(*

.. <legal notes>

legal notes
=================
| SPDX-FileCopyrightText: © 2025 Oleksandr Tiutyk <trofimich@gmail.com>
| SPDX-License-Identifier: LGPL-3.0-only
| For details check: LGPL-3.0-only_

.. _LGPL-3.0-only: https://www.gnu.org/licenses/lgpl-3.0.en.html

.. </legal notes>

*)

{attribute 'no_explicit_call' := 'do not call this function block directly'} 
FUNCTION_BLOCK DeleteDirectory EXTENDS TOF_Tasks.Task IMPLEMENTS IFileSystemTask
VAR
	_ClassName : STRING := __POUNAME();

    _DeleteDirectory : Tc2_System.FB_RemoveDir;	
END_VAR

{attribute 'monitoring' := 'call'}
PROPERTY AmsNetId : Tc2_System.T_AmsNetID
GET
AmsNetId := _DeleteDirectory.sNetId;
END_GET
SET
_DeleteDirectory.sNetId := AmsNetId;
END_SET
END_PROPERTY

{attribute 'monitoring' := 'call'}
PROPERTY ClassName : STRING
GET
ClassName := _ClassName;
END_GET
END_PROPERTY

{attribute 'monitoring' := 'call'}
PROPERTY DirectoryPath : Tc2_System.T_MaxString
GET
DirectoryPath := _DeleteDirectory.sPathName;
END_GET
SET
_DeleteDirectory.sPathName := DirectoryPath;
END_SET
END_PROPERTY

{attribute 'monitoring' := 'call'}
PROPERTY NamespaceName : STRING
GET
NamespaceName := CurrentNamespace.Name;
END_GET
END_PROPERTY

METHOD PROTECTED OnCancel
_DeleteDirectory(bExecute := FALSE);
END_METHOD

METHOD PROTECTED OnRunning 
VAR_INPUT
	startRequest : BOOL;
END_VAR
VAR_OUTPUT
	state : TASK_RUNNING_STATE;
END_VAR
VAR
	propertyNotSpecifiedException :	TOF_Core.DataMemberNotSpecifiedException;
	invalidPathException : InvalidPathException;	
	deleteDirectoryException : TOF_Core.StandardException;
	
	pathErrorMessage : WSTRING(255);
	errorMessageBuilder : TOF_Core.WideStringBuilder;
END_VAR
IF startRequest THEN 
	IF TOF_Core.StringHelper.IsNullOrWhiteSpace(_DeleteDirectory.sPathName) THEN
		propertyNotSpecifiedException.Throw(NamespaceName, ClassName, __POUNAME(), __POSITION(), 'DirectoryPath');		
	END_IF
	
	IF NOT PathHelper.IsValidDirectoryPath(_DeleteDirectory.sPathName, errorMessage => pathErrorMessage) THEN
		invalidPathException.Throw(NamespaceName, ClassName, __POUNAME(), __POSITION(), _DeleteDirectory.sPathName, pathErrorMessage);
	END_IF
	
	_DeleteDirectory(bExecute := FALSE);
END_IF

_DeleteDirectory(bExecute := TRUE);

IF _DeleteDirectory.bError THEN
	errorMessageBuilder
		.AppendString("An error occurred while deleting the directory '")
		.Append(_DeleteDirectory.sPathName)
		.AppendString("'");

	deleteDirectoryException.Throw(NamespaceName, ClassName, __POUNAME(), __POSITION(), errorMessageBuilder.ToString255(), errorCode := _DeleteDirectory.nErrId);
END_IF

IF NOT _DeleteDirectory.bBusy THEN
	state := TOF_Tasks.TASK_RUNNING_STATE.DONE;
END_IF
END_METHOD

{attribute 'monitoring' := 'call'}
PROPERTY PathType : Tc2_System.E_OpenPath
GET
PathType := _DeleteDirectory.ePath;
END_GET
SET
_DeleteDirectory.ePath := PathType;
END_SET
END_PROPERTY

{attribute 'monitoring' := 'call'}
PROPERTY Size : ULINT
GET
Size := XSIZEOF(THIS^);
END_GET
END_PROPERTY

{attribute 'monitoring' := 'call'}
PROPERTY Timeout : TIME
GET
Timeout := _DeleteDirectory.tTimeout;
END_GET
SET
_DeleteDirectory.tTimeout := Timeout;
END_SET
END_PROPERTY

END_FUNCTION_BLOCK

(* stored: Version 1.1.0.1
   POU DeleteDirectory: Id {f7699339-eb16-4c49-8ff9-e8b510a181bf}, SpecialFunc None
   Folder Inputs: Id {3c1b2bb2-508a-43ab-aba6-d51610d36987}
   Folder Members to override: Id {80e81cc0-48cb-4c8d-a6d2-f5019c2649ac}
   Property AmsNetId: Id {e619447a-91f5-4cfd-87c1-c6f4d65469a7}
   Get Get: Id {af838fb5-84a9-40c2-96ed-bb37e1ba8ee8}
   Set Set: Id {955f8a77-cfbb-437a-a3ea-c4c2072c8db2}
   Property ClassName: Id {9bdfd013-5a24-4a24-9847-b8d276cbdfd1}
   Get Get: Id {07f43309-f5f9-4714-8a79-b20e37081f91}
   Property DirectoryPath: Id {d94128c9-a1f4-40bf-a870-d7916c828353}
   Get Get: Id {1f72f3d7-a990-4668-a6c3-c54f2f298ded}
   Set Set: Id {39cb2b34-0284-49a9-954b-190ef76241ef}
   Property NamespaceName: Id {c30ceec4-6b12-4987-9c9a-253d7cedcfe2}
   Get Get: Id {5de19f01-2439-4806-bb38-5c646f83ed28}
   Method OnCancel: Id {854891df-525d-4ee7-8081-b1a0fedc87ce}
   Method OnRunning: Id {df915afb-aa65-445f-a579-78975326fa79}
   Property PathType: Id {2b9d54ab-fa46-41da-ac42-cdc7d5acef43}
   Get Get: Id {6baf4074-7f57-4b46-a346-9359d4fc170d}
   Set Set: Id {7a03c98f-e798-4494-b934-37bb17268ced}
   Property Size: Id {9adbdd4e-26f1-45e1-9314-6ac5a9fcf883}
   Get Get: Id {7af252a4-6350-4943-9c1e-b0b9f893fccd}
   Property Timeout: Id {c5f42126-d467-415e-a93a-fa9d11d77a43}
   Get Get: Id {3464bdc4-4947-406d-8d6a-94c7e64bc5b4}
   Set Set: Id {67cf6448-3dc3-4665-a07b-57b154ad6605} *)
